FUNCTION_BLOCK FB_Transport
VAR_INPUT
	bEnable :BOOL;
	bExecute :BOOL;
	nStation :INT;
	//Hardweare Eingänge
	bSens1 :BOOL;
	bSens2 :BOOL;
	bSens3 :BOOL;
	bSens4 :BOOL;
END_VAR
VAR_OUTPUT
	eState :eBetriebszustand;
	bStopper1 :BOOL;
	bStopper2 :BOOL;
	bStopper3 :BOOL;
END_VAR
VAR
	fb_TransportE :FB_Transport_E;
	fb_TransportLogik :FB_Transport_Logik;
	fb_TransportBand :FB_Foerderband;
	fb_TransportA :FB_Transport_A;
END_VAR
VAR_IN_OUT
	//Achsen Ref
	ax : AXIS_REF;
END_VAR

//nur Eingänge werden beschreiben 
fb_TransportE(
	bSens1:= bSens1, 
	bSens2:= bSens2, 
	bSens3:= bSens3, 
	bSens4:= bSens4, 
	bStation1=> , 
	bStation2=> , 
	bStation3=> , 
	bStation4=> );
	
fb_TransportLogik(
	bEnable:= bEnable, 
	bExecute:= bExecute, 
	eStateE:= fb_TransportBand.eState, 
	nStation:= nStation, 
	bStation1:= fb_TransportE.bStation1, 
	bStation2:= fb_TransportE.bStation2, 
	bStation3:= fb_TransportE.bStation3, 
	bEnableA=> , 
	bExecuteA=> , 
	bStopA=> , 
	eStateA=> , 
	bStop1=> , 
	bStop2=> , 
	bStop3=> );
	
	
fb_TransportBand(
	bEnable:= fb_TransportLogik.bEnableA, 
	bExecute:= fb_TransportLogik.bExecuteA, 
	bHalt:= fb_TransportLogik.bStopA, 
	eState=> , 
	ax:= ax);
	
	
fb_TransportA(
	bStop1:= fb_TransportLogik.bStop1, 
	bStop2:= fb_TransportLogik.bStop2, 
	bStop3:= fb_TransportLogik.bStop3, 
	bStopper1=> bStopper1, 
	bStopper2=> bStopper1, 
	bStopper3=> bStopper1);

END_FUNCTION_BLOCK

(* stored: Version 1.1.0.1, ProductVersion 3.1.4024.15
   POU FB_Transport: Id {326665c8-b6b7-4475-a44b-2dee740fc7ea}, SpecialFunc None *)
